Omron CX-Programmer project NewProject (CX-Programmer 9.75)

# PLC TimerTraffic: CP1E N30

## Global symbols (name address type ; comment)
T000 BOOL  ; T0
T001 BOOL  ; T1
T002 BOOL  ; T2
Red 100.01 BOOL  ; 100.01

## Program NewProgram1 (cyclic task 0)
Local symbols
Green 100.03 BOOL  ; 100.03
MainSupply 100.00 BOOL  ; 100.00
Start 0.00 BOOL  ; 0.00
Stop 0.01 BOOL  ; 0.01
Yellow 100.02 BOOL  ; 100.02

### Section Section1

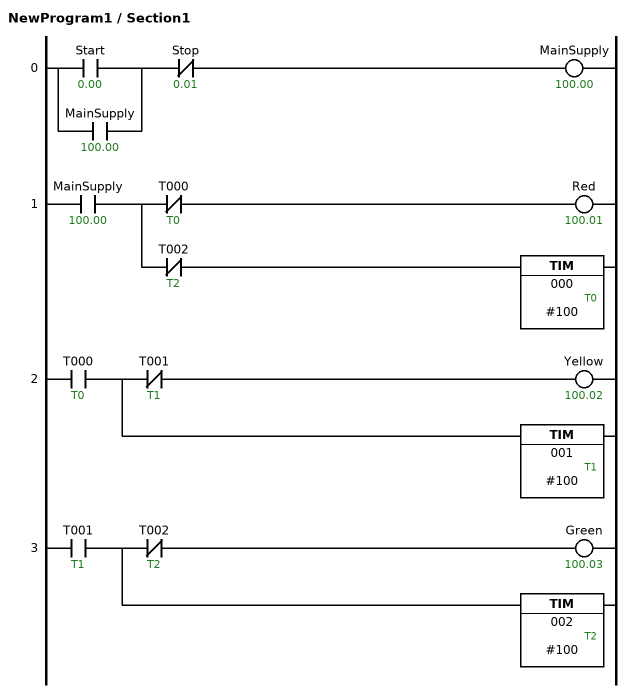
; rung 0
LD Start  ; 0.00
OR MainSupply  ; 100.00
ANDNOT Stop  ; 0.01
OUT MainSupply  ; 100.00
; rung 1
LD MainSupply  ; 100.00
OUT TR0
ANDNOT T000  ; T0
OUT Red  ; 100.01
LD TR0
ANDNOT T002  ; T2
TIM 000 #100  ; T0
; rung 2
LD T000  ; T0
OUT TR0
ANDNOT T001  ; T1
OUT Yellow  ; 100.02
LD TR0
TIM 001 #100  ; T1
; rung 3
LD T001  ; T1
OUT TR0
ANDNOT T002  ; T2
OUT Green  ; 100.03
LD TR0
TIM 002 #100  ; T2

### Section END
; rung 0
END(001)